// TIA Portal V20 export
FUNCTION "Block_4" : Void   // FC4, STL
{ S7_Optimized_Access := 'TRUE' }
BEGIN

NETWORK
TITLE = 
      A     "Switch 1 ON";
      =     "Lamp 1 ON";
END_FUNCTION
